(*
SPDX-FileCopyrightText: © 2026 Oleksandr Tiutyk <trofimich@gmail.com>
SPDX-License-Identifier: MIT
License: https://opensource.org/license/mit
*)

(*!
<summary>Provides indexed access and searching without operations that change list entries or their order.</summary>
<description>
This interface does not expose insertion, removal, replacement or reordering. It is a view, not an immutable
snapshot: changes through another mutable reference can invalidate positions. Borrowed descriptors and payload
require the source collection to remain alive. ContainsGeneric currently defaults to releasing an owned query.
Get and FindSingle return borrowed views even when their descriptor carries IsMemoryOwner; a descriptor copy
does not transfer ownership.
</description>
*)
INTERFACE IReadOnlyList EXTENDS ICollection

(*!
<summary>Searches for a value using default generic equality.</summary>
<description>
Borrows the ANY argument during a linear search without cloning or releasing it. isObject = TRUE means a live
Object FB instance, not a pointer or interface variable. Equality exceptions propagate; callbacks that mutate
the collection can invalidate traversal.
</description>
*)
METHOD Contains : BOOL
VAR_INPUT
	value : ANY;
	isObject : BOOL := FALSE;
END_VAR
END_METHOD

(*!
<summary>Searches for an equal generic value and optionally releases the query.</summary>
<description>
Uses GENERIC_VALUE.Equals in a linear search. releaseValue defaults to TRUE: after a completed search, Release
is called on the local query copy, including on a miss. Caller-side aliases are not reset. The query must not
own storage retained by the collection. Requested release is attempted after both successful lookup and lookup
failure. Before cleanup, the original framework exception is retained and a borrowed static system exception
is cloned to preserve its code, catch point and timestamps across cleanup callbacks. The captured exception is
then propagated through ExceptionManager.Throw in the current cyclic task; native errors use the framework
SystemException representation. If capturing the system exception fails with terminal OOM, query cleanup is
still attempted and terminal OOM takes precedence. Terminal allocation state is never cleared. Release is best
effort and does not prove successful deallocation. Cleanup callbacks must not reenter collection mutation.
</description>
*)
METHOD ContainsGeneric : BOOL
VAR_INPUT
	value : TOF_Core.GENERIC_VALUE;
	releaseValue : BOOL := TRUE;
END_VAR
END_METHOD

(*!
<summary>Finds a predicate match in the requested traversal direction.</summary>
<description>
skip counts matches, not visited entries. A null predicate or no match returns FALSE; outputs are meaningful
only on TRUE. The result is borrowed even if IsMemoryOwner is TRUE. Predicate input uses AsAnyType without
preserving the explicit generic OBJECT category. Predicate exceptions propagate; callbacks must not mutate the
traversed collection.
</description>
*)
METHOD FindSingle : BOOL
VAR_INPUT
	predicate : TOF_Core.IPredicate;
	skip : UDINT := 0;
	searchDirection : TOF_Core.SEARCH_DIRECTION := TOF_Core.SEARCH_DIRECTION.FROM_BEGINNING;
END_VAR
VAR_OUTPUT
	value : TOF_Core.GENERIC_VALUE;
	index : TOF_Core.DINT_INDEX;
END_VAR
END_METHOD

(*!
<summary>Reports whether fixed-capacity storage has no free slot.</summary>
<description>
Dynamic collections report FALSE even when Length equals Capacity. This does not guarantee available heap
memory.
</description>
*)
{attribute 'monitoring' := 'call'}
PROPERTY FINAL Full : BOOL
GET
END_GET
END_PROPERTY

(*!
<summary>Borrows the descriptor at a zero-based list position.</summary>
<description>
An out-of-range index raises an exception. Returned descriptors and payload are borrowed, not clones. Do not
modify descriptor metadata or release payload through this view, even when IsMemoryOwner is TRUE. Keep the
source and borrowed storage alive; mutation or destruction can invalidate the view.
</description>
*)
METHOD Get : REFERENCE TO TOF_Core.GENERIC_VALUE
VAR_INPUT
	index : TOF_Core.DINT_INDEX;
END_VAR
END_METHOD

END_INTERFACE

(* stored: Version 1.1.0.1
   Itf IReadOnlyList: Id {2ae0731d-8d43-42f2-abee-f0660bf607da}
   Method Contains: Id {3b83f8d2-7303-4790-af34-7f74cfe4fa84}
   Method ContainsGeneric: Id {2aebd1bf-df14-401f-b6a5-5d6c199aeadd}
   Method FindSingle: Id {1b102e63-f5bc-45b5-87cf-c33b4c4088e7}
   Property Full: Id {9fe15f64-e9c9-43cf-ae85-2cbc0b5e3106}
   Get Get: Id {f2c42cc1-f16e-4a3d-b820-e4d406744411}
   Method Get: Id {f5cd9212-1ade-4b6f-92a1-97d3e216a850} *)
